FUNCTION F_NormQuat : LREAL
VAR_INPUT
    iQuat : I_Quat;
END_VAR


F_NormQuat := SQRT(F_NormSqQuat(iQuat));

END_FUNCTION

(* stored: Version 1.1.0.1
   POU F_NormQuat: Id {ac45f6af-5f3f-4ad4-9ea6-4799a1a4a160}, SpecialFunc None *)
